# EPICS autosave request: IOCs/MS_DAQ/MSApp/Db/MS_settings.req
# This file is used by autosave to determine what PVs to save (currently, autosave not used)
# It is also used by MS DAQ to determine what PVs to create

# This file contains all of the PVs used by the MS.

####################
# Energy information
####################

$(P)$(R)EnergyPVName
$(P)$(R)DcctCurrentPVName
$(P)$(R)ShutterOnePVName
$(P)$(R)ShutterTwoPVName
$(P)$(R)StopperStatusPVName

####################
# Exposure Time
####################

$(P)$(R)DetExposureTimePVName

####################
# Detector Control
####################

$(P)$(R)NImagesPVName
$(P)$(R)ImageNamePVName
$(P)$(R)ImagePathPVName
$(P)$(R)isAcquiringPVName
$(P)$(R)AcquiringPVName

####################
# Detector & IOC Management
####################

$(P)$(R)DSConfigName
$(P)$(R)DSUserConfigName
$(P)$(R)TopConfigName
$(P)$(R)PilatusServerUserConfigName
$(P)$(R)PilatusServerConfigName

####################
# Data Management
####################

$(P)$(R)DataPathConfigName
$(P)$(R)DetDataPathConfigName
$(P)$(R)TestDataPathConfigName
